// TIA Portal project "visao_cortica" (V16)

(* hardware
DEVICE "S7-1200 station_1"  S7-1200 Station
   slot 0: "Rack_0"  S7-1200 Rack  Rack  V1.0
   slot 1: "PLC_1"  CPU 1214C DC/DC/DC  6ES7 214-1AG40-0XB0  V4.4
DEVICE "GSD device_1"  GSD.Device.PN
   slot 0: "URIODev1"  V1.0  00000
      slot 0: "V1.0"  V1.0
      slot 1: "Interface"  Interface
         slot 1: "RJ45 10/100 MBit/s"  RJ45 10/100 MBit/s
   slot 0: "Rack"  Rack  V1.0
   slot 1: "1_T2O State_1"  1_T2O State  1.0
      slot 0: "1_T2O State"  1_T2O State
   slot 2: "2_T2O IO_1"  2_T2O IO  1.0
      slot 0: "2_T2O IO"  2_T2O IO
   slot 3: "3_T2O Joints_1"  3_T2O Joints  1.0
      slot 0: "3_T2O Joints"  3_T2O Joints
   slot 4: "4_T2O TCP_1"  4_T2O TCP  1.0
      slot 0: "4_T2O TCP"  4_T2O TCP
   slot 5: "5_T2O General Purpose Bit Registers_1"  5_T2O General Purpose Bit Registers  1.0
      slot 0: "5_T2O General Purpose Bit Registers"  5_T2O General Purpose Bit Registers
   slot 6: "6_T2O General Purpose Int Registers_1"  6_T2O General Purpose Int Registers  1.0
      slot 0: "6_T2O General Purpose Int Registers"  6_T2O General Purpose Int Registers
   slot 7: "7_T2O General Purpose Float Registers_1"  7_T2O General Purpose Float Registers  1.0
      slot 0: "7_T2O General Purpose Float Registers"  7_T2O General Purpose Float Registers
   slot 8: "8_O2T Robot IO_1"  8_O2T Robot IO  1.0
      slot 0: "8_O2T Robot IO"  8_O2T Robot IO
   slot 9: "9_O2T General Purpose Registers 1_1"  9_O2T General Purpose Registers 1  1.0
      slot 0: "9_O2T General Purpose Registers 1"  9_O2T General Purpose Registers 1
   slot 10: "10_O2T General Purpose Registers 2_1"  10_O2T General Purpose Registers 2  1.0
      slot 0: "10_O2T General Purpose Registers 2"  10_O2T General Purpose Registers 2
*)

// ===== PLC "PLC_1"  CPU 1214C DC/DC/DC =====

VAR_GLOBAL   // PLC tag table "Robot Tags"
   "T20_state" AT %I2.0 : "UR_1_T2O_State";
   "T20_IO" AT %I68.0 : "UR_2_T2O_IO";
   "T20_Joints" AT %I136.0 : "UR_3_T2O_Joints";
   "T20_TCP" AT %I240.0 : "UR_4_T2O_TCP";
   "T20_general_prop_bit_registers" AT %I34.0 : "UR_5_T2O_BitRegisters";
   "T20_IntRegisters" AT %I316.0 : "UR_6_T2O_IntRegisters";
   "T20_FloatRegisters" AT %I412.0 : "UR_7_T2O_FloatRegisters";
   "O2T_Robot_IO" AT %Q2.0 : "UR_8_O2T_Robot_IO";
   "O2T_General_purpose_register" AT %Q26.0 : "UR_9_O2T_Registers";
   "O2T_General_purpose_register_2" AT %Q126.0 : "UR_9_O2T_Registers";
   "Start program" AT %Q2.1 : Bool;
   "Stop program" AT %Q2.2 : Bool;
   "Pause program" AT %Q2.3 : Bool;
   "botao_start" AT %I2.1 : Bool;
   "botao_pausa" AT %I2.2 : Bool;
   "botao_stop" AT %I2.3 : Bool;
   "botao segurança" AT %I2.4 : Bool;
   "ligar" AT %I2.5 : Bool;
   "condicoes_iniciais" AT %M1.0 : Bool;
   "S1" AT %M1.2 : Bool;
   "S2" AT %M1.3 : Bool;
   "s0" AT %M1.1 : Bool;
END_VAR

TYPE "User_data_type_1"
END_TYPE

TYPE "UR__O2T_Robot"
   STRUCT
      "SSM: Speed slider fraction mask" : Bool;
      Reserved_1 : Bool;
      Reserved_2 : Bool;
      Reserved_3 : Bool;
      Reserved_4 : Bool;
      Reserved_5 : Bool;
      Reserved_6 : Bool;
      Reserved_7 : Bool;
      Reserved_8_15 : USInt;
      Reserved_16_31 : UInt;
      "Speed slider fraction" : Real;
   END_STRUCT;
END_TYPE

TYPE "UR__O2T_ints"
   STRUCT
      Register : Array[0..11] of DInt;
   END_STRUCT;
END_TYPE

TYPE "UR__O2T_floats"
   STRUCT
      Register : Array[0..11] of Real;
   END_STRUCT;
END_TYPE

TYPE "UR__O2T_IOs"
   STRUCT
      "Standard digital output mask" : USInt;
      "Configurable digital output mask" : USInt;
      "Standard digital outputs" : USInt;
      "Configurable digital outputs" : USInt;
      "AOM: Analog output mask" : USInt;
      "AOT: Analog output types" : USInt;
      "TDOM: Tool digital output mask" : USInt;
      "TDO: Tool digital output" : USInt;
      "Standard analog output" : Array[0..1] of Real;
   END_STRUCT;
END_TYPE

TYPE "UR__O2T_bits"
   STRUCT
      Register : Array[0..31] of Bool;
   END_STRUCT;
END_TYPE

TYPE "UR_9_O2T_Registers"
   STRUCT
      Bits : "UR__O2T_bits";
      Ints : "UR__O2T_ints";
      Floats : "UR__O2T_floats";
   END_STRUCT;
END_TYPE

TYPE "UR__T2O_IOs"
   STRUCT
      "Standard digital inputs" : USInt;
      "Configurable digital inputs" : USInt;
      "Standard digital outputs" : USInt;
      "Configurable digital outputs" : USInt;
      "Analog I/O types" : USInt;
      Reserved_8_15 : USInt;
      Reserved_16_31 : UInt;
      "Standard analog input [A or V]" : Array[0..1] of Real;
      "Standard analog output [A or V]" : Array[0..1] of Real;
      "I/O current [A]" : Real;
      "Euromap67 input bits" : Array[0..31] of Bool;
      "Euromap67 output bits" : Array[0..31] of Bool;
      "Euromap67 24V voltage" : Real;
      "Euromap67 24V current" : Real;
   END_STRUCT;
END_TYPE

TYPE "UR_8_O2T_Robot_IO"
   STRUCT
      Robot : "UR__O2T_Robot";
      IOs : "UR__O2T_IOs";
   END_STRUCT;
END_TYPE

TYPE "UR__T2O_Safety"
   STRUCT
      "Safety mode" : USInt;
      Reserved_1 : USInt;
      Reserved_2 : UInt;
      "NO: Is normal mode" : Bool;
      "RD: Is reduced mode" : Bool;
      "PS: Is protective stopped" : Bool;
      "RC: Is recovery mode" : Bool;
      "SS: Is safeguard stopped" : Bool;
      "SES: Is system emergency stopped" : Bool;
      "RES: Is robot emergency stopped" : Bool;
      "ES: Is emergency stopped" : Bool;
      "VL: Is violation" : Bool;
      "FT: Is fault" : Bool;
      "ST: Is stopped due to safety" : Bool;
      Reserved_11 : Bool;
      Reserved_12 : Bool;
      Reserved_13 : Bool;
      Reserved_14 : Bool;
      Reserved_15 : Bool;
      Reserved_16_31 : UInt;
   END_STRUCT;
END_TYPE

TYPE "UR__T2O_Robot"
   STRUCT
      "Controller major version" : USInt;
      "Controller minor version" : USInt;
      Reserved : UInt;
      "Robot mode" : USInt;
      "Real time machine seconds" : USInt;
      "Real time machine milliseconds" : UInt;
      "Real time machine minutes" : USInt;
      "Real time machine hours" : USInt;
      "Real time machine days" : UInt;
      "Robot current [A]" : Real;
      "PW: Is power on" : Bool;
      "PR: Is program running" : Bool;
      "TB: Is teach button pressed" : Bool;
      "PB: Is power button pressed" : Bool;
      Reserved_4 : Bool;
      Reserved_5 : Bool;
      Reserved_6 : Bool;
      Reserved_7 : Bool;
      Reserved_8_15 : USInt;
      Reserved_16_31 : UInt;
      "Speed slider fraction" : Real;
   END_STRUCT;
END_TYPE

TYPE "UR__T2O_Tool"
   STRUCT
      "Tool mode" : USInt;
      Reserved_7_15 : USInt;
      Reserved_16_31 : UInt;
      "TDI: Tool Digital Inputs" : USInt;
      "TDO: Tool Digital Outputs" : USInt;
      "TAIT: Tool Analog Input Types" : USInt;
      Reserved_24_31 : USInt;
      "Tool analog input [A or V]" : Array[0..1] of Real;
      "Tool output voltage [V]" : Real;
      "Tool current [A]" : Real;
   END_STRUCT;
END_TYPE

TYPE "UR_O2T"
   STRUCT
      "Robot IO" : "UR_8_O2T_Robot_IO";
      "Reg 1" : "UR_9_O2T_Registers";
      "Reg 2" : "UR_9_O2T_Registers";
   END_STRUCT;
END_TYPE

TYPE "UR_4_T2O_TCP"
   STRUCT
      "TCP Position (X,Y,Z) [m]" : Array[0..2] of Real;
      "TCP Position (RX,RY,RZ) [rad]" : Array[0..2] of Real;
      "TCP velocity (X,Y,Z) [m/s]" : Array[0..2] of Real;
      "TCP velocity (RX,RY,RZ) [rad/s]" : Array[0..2] of Real;
      "TCP force (X,Y,Z) [N]" : Array[0..2] of Real;
      "TCP torque (X,Y,Z) [Nm]" : Array[0..2] of Real;
      "TCP force scalar [N]" : Real;
   END_STRUCT;
END_TYPE

TYPE "UR_3_T2O_Joints"
   STRUCT
      "Joint position [rad]" : Array[0..5] of Real;
      "Joint velocity [rad/s]" : Array[0..5] of Real;
      "Joint current [A]" : Array[0..5] of Real;
      "Joint temperature [°C]" : Array[0..5] of Real;
      "Joint mode" : Array[0..5] of USInt;
      Reserved_9 : UInt;
   END_STRUCT;
END_TYPE

TYPE "UR_2_T2O_IO"
   STRUCT
      IOs : "UR__T2O_IOs";
      Tool : "UR__T2O_Tool";
   END_STRUCT;
END_TYPE

TYPE "UR_5_T2O_BitRegisters"
   STRUCT
      Register : Array[0..63] of Bool;
   END_STRUCT;
END_TYPE

TYPE "UR_1_T2O_State"
   STRUCT
      Robot : "UR__T2O_Robot";
      Safety : "UR__T2O_Safety";
   END_STRUCT;
END_TYPE

TYPE "UR_7_T2O_FloatRegisters"
   STRUCT
      Register : Array[0..23] of Real;
   END_STRUCT;
END_TYPE

TYPE "UR_6_T2O_IntRegisters"
   STRUCT
      Register : Array[0..23] of DInt;
   END_STRUCT;
END_TYPE

TYPE "UR_T2O"
   STRUCT
      State : "UR_1_T2O_State";
      IO : "UR_2_T2O_IO";
      Joints : "UR_3_T2O_Joints";
      TCP : "UR_4_T2O_TCP";
      Bits : "UR_5_T2O_BitRegisters";
      Ints : "UR_6_T2O_IntRegisters";
      Floats : "UR_7_T2O_FloatRegisters";
   END_STRUCT;
END_TYPE

FUNCTION "ur10" : Void   // FC1, LAD
{ S7_Optimized_Access := 'TRUE' }
VERSION : 0.1
BEGIN

REGION Network 1
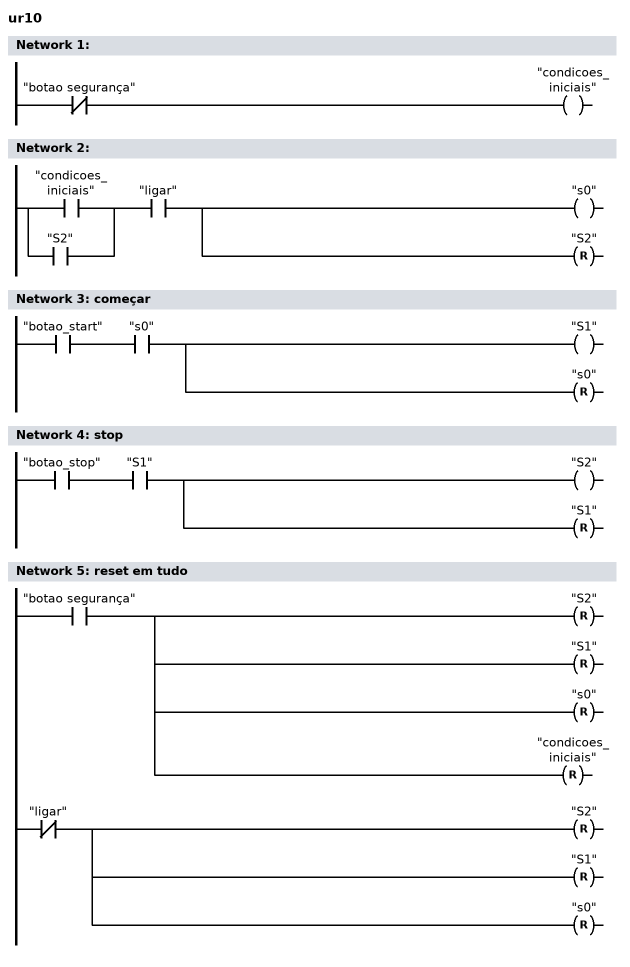
   RUNG wire#powerrail
      I_Contact( "botao segurança" )
      Coil( "condicoes_iniciais" )
   END_RUNG
   // the same network as SCL:
   "condicoes_iniciais" := NOT "botao segurança";
END_REGION

REGION Network 2
   RUNG wire#powerrail
      Contact( "condicoes_iniciais" )
      wire#w1
      Contact( "ligar" )
      wire#w2
      Coil( "s0" )
   END_RUNG
   RUNG wire#powerrail
      Contact( "S2" )
   END_RUNG wire#w1
   RUNG wire#w2
      R_Coil( "S2" )
   END_RUNG
   // the same network as SCL:
   "s0" := ("condicoes_iniciais" OR "S2") AND "ligar";
   IF "s0" THEN "S2" := FALSE; END_IF;
END_REGION

REGION Network 3: começar
   RUNG wire#powerrail
      Contact( "botao_start" )
      Contact( "s0" )
      wire#w1
      Coil( "S1" )
   END_RUNG
   RUNG wire#w1
      R_Coil( "s0" )
   END_RUNG
   // the same network as SCL:
   "S1" := "botao_start" AND "s0";
   IF "S1" THEN "s0" := FALSE; END_IF;
END_REGION

REGION Network 4: stop
   RUNG wire#powerrail
      Contact( "botao_stop" )
      Contact( "S1" )
      wire#w1
      Coil( "S2" )
   END_RUNG
   RUNG wire#w1
      R_Coil( "S1" )
   END_RUNG
   // the same network as SCL:
   "S2" := "botao_stop" AND "S1";
   IF "S2" THEN "S1" := FALSE; END_IF;
END_REGION

REGION Network 5: reset em tudo
   RUNG wire#powerrail
      Contact( "botao segurança" )
      wire#w1
      R_Coil( "S2" )
   END_RUNG
   RUNG wire#w1
      R_Coil( "S1" )
   END_RUNG
   RUNG wire#w1
      R_Coil( "s0" )
   END_RUNG
   RUNG wire#w1
      R_Coil( "condicoes_iniciais" )
   END_RUNG
   RUNG wire#powerrail
      I_Contact( "ligar" )
      wire#w2
      R_Coil( "S2" )
   END_RUNG
   RUNG wire#w2
      R_Coil( "S1" )
   END_RUNG
   RUNG wire#w2
      R_Coil( "s0" )
   END_RUNG
   // the same network as SCL:
   IF "botao segurança" THEN
       "S2" := FALSE;
       "S1" := FALSE;
       "s0" := FALSE;
       "condicoes_iniciais" := FALSE;
   END_IF;
   IF NOT "ligar" THEN
       "S2" := FALSE;
       "S1" := FALSE;
       "s0" := FALSE;
   END_IF;
END_REGION
END_FUNCTION

FUNCTION "ativaçao variaveis ur10" : Void   // FC2, LAD
{ S7_Optimized_Access := 'TRUE' }
VERSION : 0.1
BEGIN

REGION Network 1
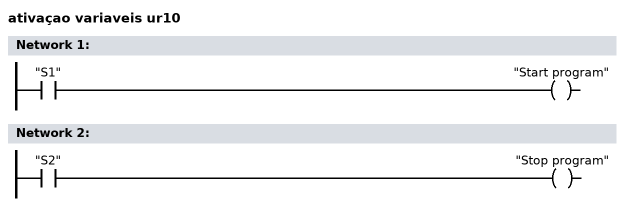
   RUNG wire#powerrail
      Contact( "S1" )
      Coil( "Start program" )
   END_RUNG
   // the same network as SCL:
   "Start program" := "S1";
END_REGION

REGION Network 2
   RUNG wire#powerrail
      Contact( "S2" )
      Coil( "Stop program" )
   END_RUNG
   // the same network as SCL:
   "Stop program" := "S2";
END_REGION
END_FUNCTION

ORGANIZATION_BLOCK "Main"   // OB1, LAD, ProgramCycle
TITLE = "Main Program Sweep (Cycle)"
{ S7_Optimized_Access := 'TRUE' }
VERSION : 0.1
   VAR_INPUT
      Initial_Call : Bool;   // Initial call of this OB
      Remanence : Bool;   // =True, if remanent data are available
   END_VAR
BEGIN
END_ORGANIZATION_BLOCK